(* LS Electric XG5000 project: 20230521 *)
(* PLC LSPLC *)

PROGRAM NewProgram (* task: 스캔 프로그램 *)
VAR
    C1 : CTU_INT;
    CTR : BOOL;
    INST : TON;
    INST1 : CTU_INT;
    INST2 : CTU_INT;
    INST3 : CTU_INT;
    P0 : BOOL;
    P1 : BOOL;
    P10 : BOOL;
    P11 : BOOL;
    P12 : BOOL;
    P2 : BOOL;
    P3 : BOOL;
    T0 : BOOL;
    T1 : BOOL;
    T2 : TON;
    T3 : TON;
    T4 : TON;
    T5 : TON;
    TF1 : TOF;
    TP1 : TP;
    TP2 : TP;
    TP3 : TP;
END_VAR
VAR
    _e1 : R_TRIG;
    _e2 : R_TRIG;
    _e3 : R_TRIG;
    _e4 : F_TRIG;
    _e5 : F_TRIG;
    _e6 : R_TRIG;
END_VAR

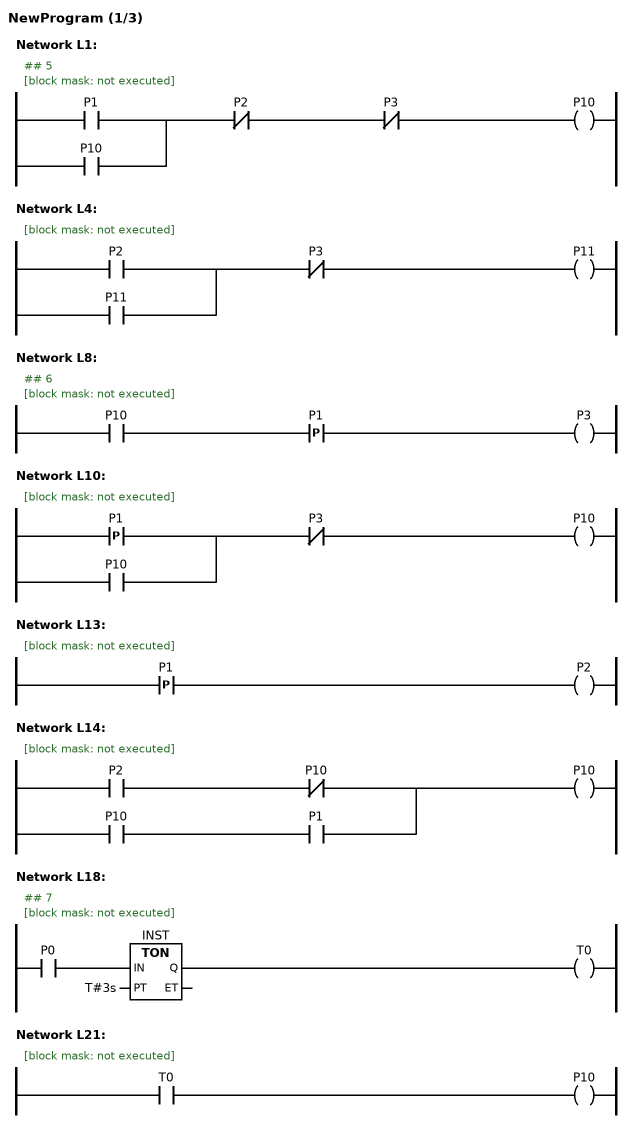
(* ## 5 *)
(* Rung L1 is block-masked: not executed *)
// P10 := (P1 OR P10) AND NOT P2 AND NOT P3;
(* Rung L4 is block-masked: not executed *)
// P11 := (P2 OR P11) AND NOT P3;
(* ## 6 *)
(* Rung L8 is block-masked: not executed *)
// _e1(CLK := P1);
// P3 := P10 AND _e1.Q;
(* Rung L10 is block-masked: not executed *)
// _e2(CLK := P1);
// P10 := (_e2.Q OR P10) AND NOT P3;
(* Rung L13 is block-masked: not executed *)
// _e3(CLK := P1);
// P2 := _e3.Q;
(* Rung L14 is block-masked: not executed *)
// P10 := (P2 AND NOT P10) OR (P10 AND P1);
(* ## 7 *)
(* Rung L18 is block-masked: not executed *)
// INST(IN := P0, PT := T#3s);
// T0 := INST.Q;
(* Rung L21 is block-masked: not executed *)
// P10 := T0;

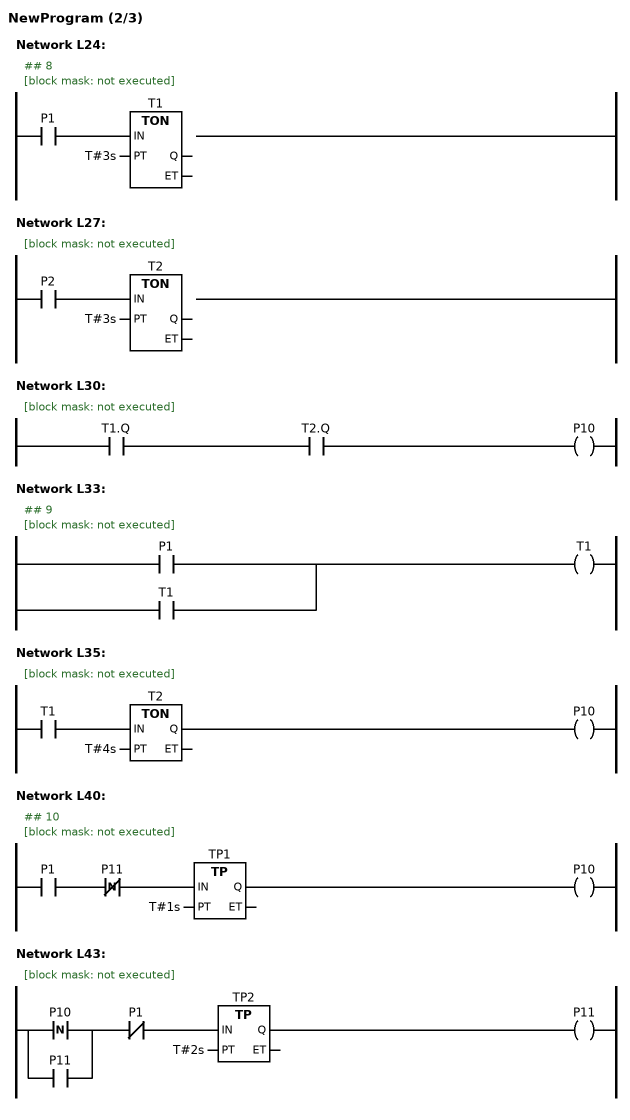
(* ## 8 *)
(* Rung L24 is block-masked: not executed *)
// T1(IN := P1, PT := T#3s);
(* Rung L27 is block-masked: not executed *)
// T2(IN := P2, PT := T#3s);
(* Rung L30 is block-masked: not executed *)
// P10 := T1.Q AND T2.Q;
(* ## 9 *)
(* Rung L33 is block-masked: not executed *)
// T1 := P1 OR T1;
(* Rung L35 is block-masked: not executed *)
// T2(IN := T1, PT := T#4s);
// P10 := T2.Q;
(* ## 10 *)
(* Rung L40 is block-masked: not executed *)
// _e4(CLK := P11);
// TP1(IN := P1 AND NOT _e4.Q, PT := T#1s);
// P10 := TP1.Q;
(* Rung L43 is block-masked: not executed *)
// _e5(CLK := P10);
// TP2(IN := (_e5.Q OR P11) AND NOT P1, PT := T#2s);
// P11 := TP2.Q;

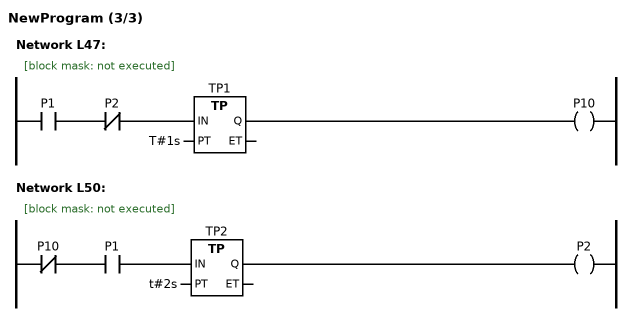
(* Rung L47 is block-masked: not executed *)
// TP1(IN := P1 AND NOT P2, PT := T#1s);
// P10 := TP1.Q;
(* Rung L50 is block-masked: not executed *)
// TP2(IN := NOT P10 AND P1, PT := t#2s);
// P2 := TP2.Q;

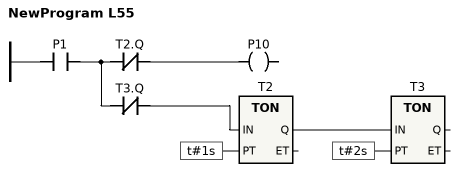
(* Rung L55 is block-masked: not executed *)
// P10 := P1 AND NOT T2.Q;
// T2(IN := P1 AND NOT T3.Q, PT := t#1s);
// T3(IN := T2.Q, PT := t#2s);

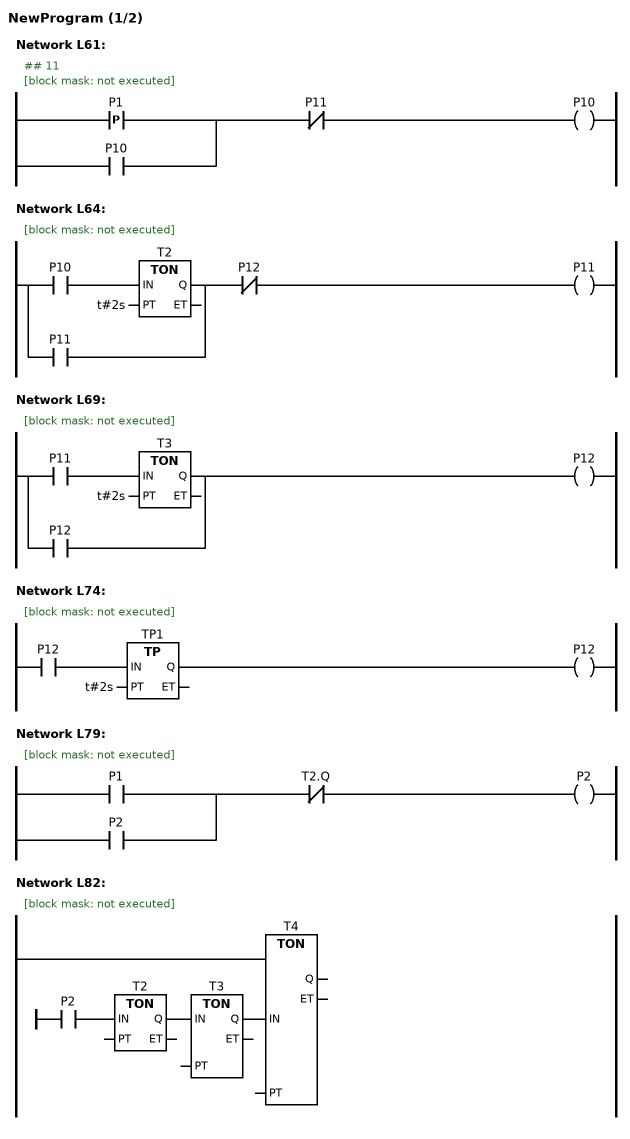
(* ## 11 *)
(* Rung L61 is block-masked: not executed *)
// _e6(CLK := P1);
// P10 := (_e6.Q OR P10) AND NOT P11;
(* Rung L64 is block-masked: not executed *)
// T2(IN := P10, PT := t#2s);
// P11 := (T2.Q OR P11) AND NOT P12;
(* Rung L69 is block-masked: not executed *)
// T3(IN := P11, PT := t#2s);
// P12 := T3.Q OR P12;
(* Rung L74 is block-masked: not executed *)
// TP1(IN := P12, PT := t#2s);
// P12 := TP1.Q;
(* Rung L79 is block-masked: not executed *)
// P2 := (P1 OR P2) AND NOT T2.Q;
(* Rung L82 is block-masked: not executed *)
// T2(IN := P2);
// T3(IN := T2.Q);
// T4(IN := T3.Q);

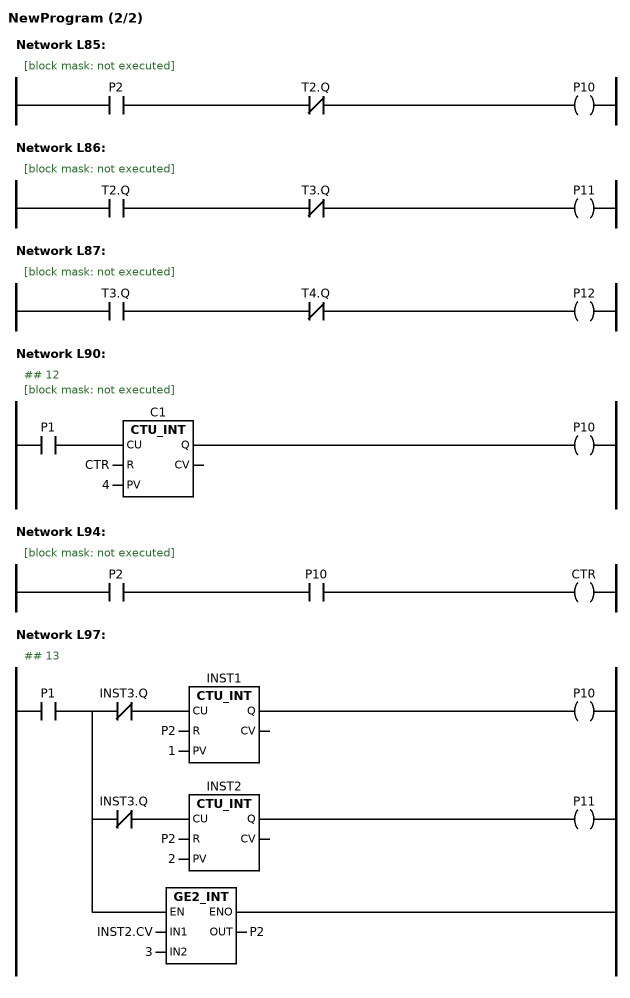
(* Rung L85 is block-masked: not executed *)
// P10 := P2 AND NOT T2.Q;
(* Rung L86 is block-masked: not executed *)
// P11 := T2.Q AND NOT T3.Q;
(* Rung L87 is block-masked: not executed *)
// P12 := T3.Q AND NOT T4.Q;
(* ## 12 *)
(* Rung L90 is block-masked: not executed *)
// C1(CU := P1, R := CTR, PV := 4);
// P10 := C1.Q;
(* Rung L94 is block-masked: not executed *)
// CTR := P2 AND P10;
(* ## 13 *)
(* Rung L97 *)
INST1(CU := P1 AND NOT INST3.Q, R := P2, PV := 1);
P10 := INST1.Q;
INST2(CU := P1 AND NOT INST3.Q, R := P2, PV := 2);
P11 := INST2.Q;
IF P1 THEN P2 := GE2_INT(INST2.CV, 3); END_IF;
END_PROGRAM